TYPE ST_P_SCREWING :
STRUCT
	PreScrewingActive:				BOOL;
	PreScrewingPrg:					INT;
	ScrewingPrg:					INT;
	PosNumber:						INT;
END_STRUCT
END_TYPE

(* stored: Version 1.1.0.1, ProductVersion 3.1.4024.10
   DUT ST_P_SCREWING: Id {1a26132c-b4c0-4da2-b231-907d78afebc3} *)
